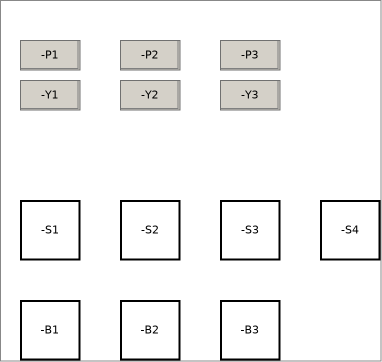
VISUALIZATION KlebeStation  // 382x362
    Button (220,40 60x30), "-P3"
        tap dSub.P3
    Button (20,80 60x30), "-Y1"
        tap dSub.Y1
    Button (120,80 60x30), "-Y2"
        tap dSub.Y2
    Button (220,80 60x30), "-Y3"
        tap dSub.Y3
    Button (20,40 60x30), "-P1"
        tap dSub.P1
    Button (120,40 60x30), "-P2"
        tap dSub.P2
    Rectangle (220,200 60x60), "-S3", colour toggle: dSub.S3
    Rectangle (320,200 60x60), "-S4", colour toggle: dSub.S4
    Rectangle (20,300 60x60), "-B1", colour toggle: dSub.B1
    Rectangle (120,300 60x60), "-B2", colour toggle: dSub.B2
    Rectangle (220,300 60x60), "-B3", colour toggle: dSub.B3
    Rectangle (20,200 60x60), "-S1", colour toggle: dSub.S1
    Rectangle (120,200 60x60), "-S2", colour toggle: dSub.S2
END_VISUALIZATION

(* stored: Version 1.1.0.1, ProductVersion 3.1.4022.6
   Visu KlebeStation: Id {529ab607-a3a7-4016-be48-cafee3caa910} *)
